PROGRAM MAIN_SQL
VAR
END_VAR

// Obsługa nowego systemu PIM
GVL.fbSqlCore(bEnable:= GVL_Aircom.bInitDone, 
	iMaxActiveNodesNb := MAIN.iMaxSimCmdNumber, 
	bKeepConnOpen := MAIN.bKeepSQLConnected, 
	iResendNbIfError:= 2,
	tCommTimeout := T#6S,
	bMasterError=> );

END_PROGRAM

(* stored: Version 1.1.0.1, ProductVersion 3.1.4024.13
   POU MAIN_SQL: Id {47b3d3cd-ccf1-479b-867b-fba47a74ead5}, SpecialFunc None *)
